(* PLC project CODEYS Common Library Template, TK TC6_v0200_Example1 v2.0, author 3S - Smart Software Solutions GmbH *)
(* stored: creationDateTime 2020-04-25T16:06:08.4861619, version 3.5.15.10, modificationDateTime 2020-04-25T16:01:39.8406952, organization 3S - Smart Software Solutions GmbH *)
(* Library project template with all possible element types, docu and a sample project structure *)

(* {attribute 'conditionalshow'} {attribute 'conditionalshow' := 'SomeText'} {attribute 'hide'} *)
{attribute 'qualified_only'}
TYPE ERROR : (NO_ERROR, TIME_OUT);
END_TYPE

{attribute 'qualified_only'}
VAR_GLOBAL CONSTANT  (* Constants - {attribute 'conditionalshow'} {attribute 'conditionalshow' := 'SomeText'} {attribute 'hide'} *)
  gc_iDummy : INT := 42;
END_VAR

{attribute 'qualified_only'}
VAR_GLOBAL  (* Variables - {attribute 'conditionalshow'} {attribute 'conditionalshow' := 'SomeText'} {attribute 'hide'} *)
  g_iDummy : INT;
END_VAR

(* {attribute 'hide_all_locals'} {attribute 'conditionalshow_all_locals' := 'SomeText'} {attribute 'conditionalshow_all_locals'} {attribute 'conditionalshow' := 'SomeText'} {attribute 'conditionalshow'} {attribute 'hide'} *)
FUNCTION_BLOCK ETrig_Temp EXTENDS CBML.ETrig
  VAR_OUTPUT
    eErrorID : ERROR;
  END_VAR

            SUPER^();
eErrorID := _Model.iErrorID;


          

METHOD CleanupAction
  VAR_INPUT
    xAbortProposed : BOOL;
    iErrorIDProposed : INT;
  END_VAR
  VAR_OUTPUT
    xComplete : BOOL := TRUE;
    xAbort : BOOL := xAbortProposed;
    iErrorID : INT := iErrorIDProposed;
  END_VAR
                  {analysis -2} 
/// ``CleanupAction`` is running until one of the following events occurs:
/// When ``xComplete`` is ``TRUE`` the state |STATE.DONE| is reached.
/// When ``xAbort`` is ``TRUE`` the state |STATE.ABORTED| is reached.
/// When ``iErrorID`` ≠ 0 (Zero) the state |STATE.ERROR| is reached.
///
/// | After a *Ready Condition* as input (``iErrorIDProposed`` = 0 and ``xAbortProposed`` = ``FALSE``), only the output states
/// | `DONE` (``xComplete`` is ``TRUE``) or `ERROR` (``iErrorID`` ≠ 0) are possible.
///
/// | After a *Error Condition* as input (``iErrorIDProposed`` ≠ 0), only the output state
/// | `ERROR` (``iErrorID`` ≠ 0) is possible.
///
/// | After a *Abort Condition* as Input (``xAbortProposed`` = ``TRUE``), only the output states
/// | `ABORTED` (``xAbort`` is ``TRUE``) or `ERROR` (``iErrorID`` ≠ 0) are possible.
///
/// .. admonition:: Example
///
///     .. code-block:: codesys
///     
///         (* common cleanup -- first steps *) 
///         
///         IF xComplete THEN
///             IF xAbortProposed THEN
///                 (* abort condition -- abort specific cleanup *)
///                 xAbort := TRUE;
///                 xComplete := FALSE;
///             ELSIF iErrorIDProposed <> 0 THEN
///                 (* error condition -- error specific cleanup *)
///                 iErrorID := SEL(xComplete, 0, iErrorIDProposed);
///                 xComplete := FALSE;
///             ELSE
///                 (* ready condition -- done specific cleanup*)
///             END_IF
///         END_IF
///
///         (* common cleanup -- last steps *) 
///
/// .. note::
///
///    If this method will not provide any implementation, please remove it!

                
END_METHOD

METHOD CyclicAction
  VAR_INPUT
    itfTimingController : CBML.ITimingController;
  END_VAR
  VAR_OUTPUT
    xComplete : BOOL := TRUE;
    iErrorID : INT := 0;
  END_VAR
                  {analysis -2} 
/// The CyclicAction is running until either ``xComplete`` is ``TRUE`` or ``iErrorID`` ≠  0 (Zero).
/// If ``xComplete`` is ``TRUE`` or ``iErrorID`` ≠  0 (Zero) the state |STATE.CLEANING| is reached.
/// With ``itfTimingController`` ≠  0 (Zero) it is possible to check the current invocation time (see: |ITimingController.ControllerCheckTiming|).
/// Function blocks with a ``udiTimeLimit`` input variable (see: |IETrigTl|, |IETrigATl|, |IETrigTlTo|, |IETrigATlTo|, |ILConTl|, |ILConTlTo|, |ILConTlC|)
/// should be implement in such a way that the current invocation is exited when the consumed time for this invocation has exceeded the settings from udiTimeLimit.
///
/// .. admonition:: Example
///
///     .. code-block:: codesys
///     
///         REPEAT
///             // working to reach the ready condition
///             // ⇒ xComplete := TRUE
///             // if the maximum invocation time is reached
///             // ⇒ xTimeLimit := TRUE
///             // if the maximum operating time is reached
///             // ⇒ xTimeOut := TRUE
///             // if an error condition is reached
///             // ⇒ set iErrorID to a value other than 0 (Zero)
///             itfTimingController.ControllerCheckTiming(
///                 xTimeOut=>xTimeOut,
///                 xTimeLimit=>xTimeLimit
///             );
///         
///             xComplete := TRUE;
///             iErrorID := ERROR.NO_ERROR;
///     
///         UNTIL xComplete OR
///               xTimeOut OR xTimeLimit OR
///               iErrorID <> ERROR.NO_ERROR
///         END_REPEAT
///
/// .. note::
///
///    If this method will not provide any implementation, please remove it!

                
END_METHOD

METHOD ExitAction
  VAR_INPUT
    xAfterCleanup : BOOL;
    xInCopyCode : BOOL;
  END_VAR
                  {analysis -2} 
/// This method is intended for releasing external resources (like RTS handles).
/// Do not call other internal function block instances in the context of this method.
/// Call only external functions defined inside the RTS.
/// For cleaning up other resources then external ones, please use the ``CleanupAction``.
/// This method should be callable in the context of ``FB_EXIT`` for example
/// before downloading a new application or before reseting an application.
///
/// .. note::
///
///    If this method will not provide any implementation, please remove it!

                
END_METHOD

METHOD ResetAction
  VAR_OUTPUT
    xComplete : BOOL := TRUE;
  END_VAR
                  {analysis -2} 
/// The ``ResetAction`` is running until the output ``xComplete`` is ``TRUE``.
/// If ``xComplete`` is ``TRUE`` the state |STATE.DORMANT| is reached.
///
/// .. note::
///
///    If this method will not provide any implementation, please remove it!

                
END_METHOD

METHOD SampleAction
  VAR_OUTPUT
    iErrorID : INT := 0;
  END_VAR
                  {analysis -2} 
/// After leaving the state |STATE.DORMANT| the ``SampleAction`` is running one time then the state |STATE.STARTING| is reached.
/// If there is a ``iErrorID`` ≠  0 (Zero) the state |STATE.CLEANING| is reached instead.
///
/// .. note::
///
///    If this method will not provide any implementation, please remove it!

                
END_METHOD

METHOD StartAction
  VAR_OUTPUT
    xComplete : BOOL := TRUE;
    iErrorID : INT := 0;
  END_VAR
                  {analysis -2} 
/// The ``StartAction`` is running until either the output ``xComplete`` is ``TRUE`` or ``iErrorID`` ≠ 0 (Zero).
/// If ``xComplete`` is ``TRUE`` the state |STATE.EXECUTING| is reached.
/// If there is a ``iErrorID`` ≠  0 (Zero) the state |STATE.CLEANING| is reached.
///
/// .. note::
///
///    To sample the inputs in the first invocation of a function block the method SampleAction is the solution of choice.
///    See: |ISampleActionProvider.SampleAction|
///
/// .. note::
///
///    If this method will not provide any implementation, please remove it!

                
END_METHOD
END_FUNCTION_BLOCK

(* {attribute 'hide_all_locals'} {attribute 'conditionalshow_all_locals' := 'SomeText'} {attribute 'conditionalshow_all_locals'} {attribute 'conditionalshow' := 'SomeText'} {attribute 'conditionalshow'} {attribute 'hide'} *)
FUNCTION_BLOCK ETrigA_Temp EXTENDS CBML.ETrigA
  VAR_OUTPUT
    eErrorID : ERROR;
  END_VAR

            SUPER^();
eErrorID := _Model.iErrorID;

          

METHOD CleanupAction
  VAR_INPUT
    xAbortProposed : BOOL;
    iErrorIDProposed : INT;
  END_VAR
  VAR_OUTPUT
    xComplete : BOOL := TRUE;
    xAbort : BOOL := xAbortProposed;
    iErrorID : INT := iErrorIDProposed;
  END_VAR
                  {analysis -2} 
/// ``CleanupAction`` is running until one of the following events occurs:
/// When ``xComplete`` is ``TRUE`` the state |STATE.DONE| is reached.
/// When ``xAbort`` is ``TRUE`` the state |STATE.ABORTED| is reached.
/// When ``iErrorID`` ≠ 0 (Zero) the state |STATE.ERROR| is reached.
///
/// | After a *Ready Condition* as input (``iErrorIDProposed`` = 0 and ``xAbortProposed`` = ``FALSE``), only the output states
/// | `DONE` (``xComplete`` is ``TRUE``) or `ERROR` (``iErrorID`` ≠ 0) are possible.
///
/// | After a *Error Condition* as input (``iErrorIDProposed`` ≠ 0), only the output state
/// | `ERROR` (``iErrorID`` ≠ 0) is possible.
///
/// | After a *Abort Condition* as Input (``xAbortProposed`` = ``TRUE``), only the output states
/// | `ABORTED` (``xAbort`` is ``TRUE``) or `ERROR` (``iErrorID`` ≠ 0) are possible.
///
/// .. admonition:: Example
///
///     .. code-block:: codesys
///     
///         (* common cleanup -- first steps *) 
///         
///         IF xComplete THEN
///             IF xAbortProposed THEN
///                 (* abort condition -- abort specific cleanup *)
///                 xAbort := TRUE;
///                 xComplete := FALSE;
///             ELSIF iErrorIDProposed <> 0 THEN
///                 (* error condition -- error specific cleanup *)
///                 iErrorID := SEL(xComplete, 0, iErrorIDProposed);
///                 xComplete := FALSE;
///             ELSE
///                 (* ready condition -- done specific cleanup*)
///             END_IF
///         END_IF
///
///         (* common cleanup -- last steps *) 
///
/// .. note::
///
///    If this method will not provide any implementation, please remove it!

                
END_METHOD

METHOD CyclicAction
  VAR_INPUT
    itfTimingController : CBML.ITimingController;
  END_VAR
  VAR_OUTPUT
    xComplete : BOOL := TRUE;
    iErrorID : INT := 0;
  END_VAR
                  {analysis -2} 
/// The CyclicAction is running until either ``xComplete`` is ``TRUE`` or ``iErrorID`` ≠  0 (Zero).
/// If ``xComplete`` is ``TRUE`` or ``iErrorID`` ≠  0 (Zero) the state |STATE.CLEANING| is reached.
/// With ``itfTimingController`` ≠  0 (Zero) it is possible to check the current invocation time (see: |ITimingController.ControllerCheckTiming|).
/// Function blocks with a ``udiTimeLimit`` input variable (see: |IETrigTl|, |IETrigATl|, |IETrigTlTo|, |IETrigATlTo|, |ILConTl|, |ILConTlTo|, |ILConTlC|)
/// should be implement in such a way that the current invocation is exited when the consumed time for this invocation has exceeded the settings from udiTimeLimit.
///
/// .. admonition:: Example
///
///     .. code-block:: codesys
///     
///         REPEAT
///             // working to reach the ready condition
///             // ⇒ xComplete := TRUE
///             // if the maximum invocation time is reached
///             // ⇒ xTimeLimit := TRUE
///             // if the maximum operating time is reached
///             // ⇒ xTimeOut := TRUE
///             // if an error condition is reached
///             // ⇒ set iErrorID to a value other than 0 (Zero)
///             itfTimingController.ControllerCheckTiming(
///                 xTimeOut=>xTimeOut,
///                 xTimeLimit=>xTimeLimit
///             );
///         
///             xComplete := TRUE;
///             iErrorID := ERROR.NO_ERROR;
///     
///         UNTIL xComplete OR
///               xTimeOut OR xTimeLimit OR
///               iErrorID <> ERROR.NO_ERROR
///         END_REPEAT
///
/// .. note::
///
///    If this method will not provide any implementation, please remove it!

                
END_METHOD

METHOD ExitAction
  VAR_INPUT
    xAfterCleanup : BOOL;
    xInCopyCode : BOOL;
  END_VAR
                  {analysis -2} 
/// This method is intended for releasing external resources (like RTS handles).
/// Do not call other internal function block instances in the context of this method.
/// Call only external functions defined inside the RTS.
/// For cleaning up other resources then external ones, please use the ``CleanupAction``.
/// This method should be callable in the context of ``FB_EXIT`` for example
/// before downloading a new application or before reseting an application.
///
/// .. note::
///
///    If this method will not provide any implementation, please remove it!

                
END_METHOD

METHOD ResetAction
  VAR_OUTPUT
    xComplete : BOOL := TRUE;
  END_VAR
                  {analysis -2} 
/// The ``ResetAction`` is running until the output ``xComplete`` is ``TRUE``.
/// If ``xComplete`` is ``TRUE`` the state |STATE.DORMANT| is reached.
///
/// .. note::
///
///    If this method will not provide any implementation, please remove it!

                
END_METHOD

METHOD SampleAction
  VAR_OUTPUT
    iErrorID : INT := 0;
  END_VAR
                  {analysis -2} 
/// After leaving the state |STATE.DORMANT| the ``SampleAction`` is running one time then the state |STATE.STARTING| is reached.
/// If there is a ``iErrorID`` ≠  0 (Zero) the state |STATE.CLEANING| is reached instead.
///
/// .. note::
///
///    If this method will not provide any implementation, please remove it!

                
END_METHOD

METHOD StartAction
  VAR_OUTPUT
    xComplete : BOOL := TRUE;
    iErrorID : INT := 0;
  END_VAR
                  {analysis -2} 
/// The ``StartAction`` is running until either the output ``xComplete`` is ``TRUE`` or ``iErrorID`` ≠ 0 (Zero).
/// If ``xComplete`` is ``TRUE`` the state |STATE.EXECUTING| is reached.
/// If there is a ``iErrorID`` ≠  0 (Zero) the state |STATE.CLEANING| is reached.
///
/// .. note::
///
///    To sample the inputs in the first invocation of a function block the method SampleAction is the solution of choice.
///    See: |ISampleActionProvider.SampleAction|
///
/// .. note::
///
///    If this method will not provide any implementation, please remove it!

                
END_METHOD
END_FUNCTION_BLOCK

(* {attribute 'hide_all_locals'} {attribute 'conditionalshow_all_locals' := 'SomeText'} {attribute 'conditionalshow_all_locals'} {attribute 'conditionalshow' := 'SomeText'} {attribute 'conditionalshow'} {attribute 'hide'} *)
FUNCTION_BLOCK ETrigATl_Temp EXTENDS CBML.ETrigATl
  VAR_OUTPUT
    eErrorID : ERROR;
  END_VAR

            SUPER^();
eErrorID := _Model.iErrorID;

          

METHOD CleanupAction
  VAR_INPUT
    xAbortProposed : BOOL;
    iErrorIDProposed : INT;
  END_VAR
  VAR_OUTPUT
    xComplete : BOOL := TRUE;
    xAbort : BOOL := xAbortProposed;
    iErrorID : INT := iErrorIDProposed;
  END_VAR
                  {analysis -2} 
/// ``CleanupAction`` is running until one of the following events occurs:
/// When ``xComplete`` is ``TRUE`` the state |STATE.DONE| is reached.
/// When ``xAbort`` is ``TRUE`` the state |STATE.ABORTED| is reached.
/// When ``iErrorID`` ≠ 0 (Zero) the state |STATE.ERROR| is reached.
///
/// | After a *Ready Condition* as input (``iErrorIDProposed`` = 0 and ``xAbortProposed`` = ``FALSE``), only the output states
/// | `DONE` (``xComplete`` is ``TRUE``) or `ERROR` (``iErrorID`` ≠ 0) are possible.
///
/// | After a *Error Condition* as input (``iErrorIDProposed`` ≠ 0), only the output state
/// | `ERROR` (``iErrorID`` ≠ 0) is possible.
///
/// | After a *Abort Condition* as Input (``xAbortProposed`` = ``TRUE``), only the output states
/// | `ABORTED` (``xAbort`` is ``TRUE``) or `ERROR` (``iErrorID`` ≠ 0) are possible.
///
/// .. admonition:: Example
///
///     .. code-block:: codesys
///     
///         (* common cleanup -- first steps *) 
///         
///         IF xComplete THEN
///             IF xAbortProposed THEN
///                 (* abort condition -- abort specific cleanup *)
///                 xAbort := TRUE;
///                 xComplete := FALSE;
///             ELSIF iErrorIDProposed <> 0 THEN
///                 (* error condition -- error specific cleanup *)
///                 iErrorID := SEL(xComplete, 0, iErrorIDProposed);
///                 xComplete := FALSE;
///             ELSE
///                 (* ready condition -- done specific cleanup*)
///             END_IF
///         END_IF
///
///         (* common cleanup -- last steps *) 
///
/// .. note::
///
///    If this method will not provide any implementation, please remove it!

                
END_METHOD

METHOD CyclicAction
  VAR_INPUT
    itfTimingController : CBML.ITimingController;
  END_VAR
  VAR_OUTPUT
    xComplete : BOOL := TRUE;
    iErrorID : INT := 0;
  END_VAR
                  {analysis -2} 
/// The CyclicAction is running until either ``xComplete`` is ``TRUE`` or ``iErrorID`` ≠  0 (Zero).
/// If ``xComplete`` is ``TRUE`` or ``iErrorID`` ≠  0 (Zero) the state |STATE.CLEANING| is reached.
/// With ``itfTimingController`` ≠  0 (Zero) it is possible to check the current invocation time (see: |ITimingController.ControllerCheckTiming|).
/// Function blocks with a ``udiTimeLimit`` input variable (see: |IETrigTl|, |IETrigATl|, |IETrigTlTo|, |IETrigATlTo|, |ILConTl|, |ILConTlTo|, |ILConTlC|)
/// should be implement in such a way that the current invocation is exited when the consumed time for this invocation has exceeded the settings from udiTimeLimit.
///
/// .. admonition:: Example
///
///     .. code-block:: codesys
///     
///         REPEAT
///             // working to reach the ready condition
///             // ⇒ xComplete := TRUE
///             // if the maximum invocation time is reached
///             // ⇒ xTimeLimit := TRUE
///             // if the maximum operating time is reached
///             // ⇒ xTimeOut := TRUE
///             // if an error condition is reached
///             // ⇒ set iErrorID to a value other than 0 (Zero)
///             itfTimingController.ControllerCheckTiming(
///                 xTimeOut=>xTimeOut,
///                 xTimeLimit=>xTimeLimit
///             );
///         
///             xComplete := TRUE;
///             iErrorID := ERROR.NO_ERROR;
///     
///         UNTIL xComplete OR
///               xTimeOut OR xTimeLimit OR
///               iErrorID <> ERROR.NO_ERROR
///         END_REPEAT
///
/// .. note::
///
///    If this method will not provide any implementation, please remove it!

                
END_METHOD

METHOD ExitAction
  VAR_INPUT
    xAfterCleanup : BOOL;
    xInCopyCode : BOOL;
  END_VAR
                  {analysis -2} 
/// This method is intended for releasing external resources (like RTS handles).
/// Do not call other internal function block instances in the context of this method.
/// Call only external functions defined inside the RTS.
/// For cleaning up other resources then external ones, please use the ``CleanupAction``.
/// This method should be callable in the context of ``FB_EXIT`` for example
/// before downloading a new application or before reseting an application.
///
/// .. note::
///
///    If this method will not provide any implementation, please remove it!

                
END_METHOD

METHOD ResetAction
  VAR_OUTPUT
    xComplete : BOOL := TRUE;
  END_VAR
                  {analysis -2} 
/// The ``ResetAction`` is running until the output ``xComplete`` is ``TRUE``.
/// If ``xComplete`` is ``TRUE`` the state |STATE.DORMANT| is reached.
///
/// .. note::
///
///    If this method will not provide any implementation, please remove it!

                
END_METHOD

METHOD SampleAction
  VAR_OUTPUT
    iErrorID : INT := 0;
  END_VAR
                  {analysis -2} 
/// After leaving the state |STATE.DORMANT| the ``SampleAction`` is running one time then the state |STATE.STARTING| is reached.
/// If there is a ``iErrorID`` ≠  0 (Zero) the state |STATE.CLEANING| is reached instead.
///
/// .. note::
///
///    If this method will not provide any implementation, please remove it!

                
END_METHOD

METHOD StartAction
  VAR_OUTPUT
    xComplete : BOOL := TRUE;
    iErrorID : INT := 0;
  END_VAR
                  {analysis -2} 
/// The ``StartAction`` is running until either the output ``xComplete`` is ``TRUE`` or ``iErrorID`` ≠ 0 (Zero).
/// If ``xComplete`` is ``TRUE`` the state |STATE.EXECUTING| is reached.
/// If there is a ``iErrorID`` ≠  0 (Zero) the state |STATE.CLEANING| is reached.
///
/// .. note::
///
///    To sample the inputs in the first invocation of a function block the method SampleAction is the solution of choice.
///    See: |ISampleActionProvider.SampleAction|
///
/// .. note::
///
///    If this method will not provide any implementation, please remove it!

                
END_METHOD
END_FUNCTION_BLOCK

(* {attribute 'hide_all_locals'} {attribute 'conditionalshow_all_locals' := 'SomeText'} {attribute 'conditionalshow_all_locals'} {attribute 'conditionalshow' := 'SomeText'} {attribute 'conditionalshow'} {attribute 'hide'} *)
FUNCTION_BLOCK ETrigATlTo_Temp EXTENDS CBML.ETrigATlTo
  VAR_OUTPUT
    eErrorID : ERROR;  (* specific Outputs *)
  END_VAR

            SUPER^();
IF _Model.iErrorID = CBML.ERROR.TIME_OUT THEN
	eErrorID := ERROR.TIME_OUT;
ELSE
	eErrorID := _Model.iErrorID;
END_IF

          

METHOD CleanupAction
  VAR_INPUT
    xAbortProposed : BOOL;
    iErrorIDProposed : INT;
  END_VAR
  VAR_OUTPUT
    xComplete : BOOL := TRUE;
    xAbort : BOOL := xAbortProposed;
    iErrorID : INT := iErrorIDProposed;
  END_VAR
                  {analysis -2} 
/// ``CleanupAction`` is running until one of the following events occurs:
/// When ``xComplete`` is ``TRUE`` the state |STATE.DONE| is reached.
/// When ``xAbort`` is ``TRUE`` the state |STATE.ABORTED| is reached.
/// When ``iErrorID`` ≠ 0 (Zero) the state |STATE.ERROR| is reached.
///
/// | After a *Ready Condition* as input (``iErrorIDProposed`` = 0 and ``xAbortProposed`` = ``FALSE``), only the output states
/// | `DONE` (``xComplete`` is ``TRUE``) or `ERROR` (``iErrorID`` ≠ 0) are possible.
///
/// | After a *Error Condition* as input (``iErrorIDProposed`` ≠ 0), only the output state
/// | `ERROR` (``iErrorID`` ≠ 0) is possible.
///
/// | After a *Abort Condition* as Input (``xAbortProposed`` = ``TRUE``), only the output states
/// | `ABORTED` (``xAbort`` is ``TRUE``) or `ERROR` (``iErrorID`` ≠ 0) are possible.
///
/// .. admonition:: Example
///
///     .. code-block:: codesys
///     
///         (* common cleanup -- first steps *) 
///         
///         IF xComplete THEN
///             IF xAbortProposed THEN
///                 (* abort condition -- abort specific cleanup *)
///                 xAbort := TRUE;
///                 xComplete := FALSE;
///             ELSIF iErrorIDProposed <> 0 THEN
///                 (* error condition -- error specific cleanup *)
///                 iErrorID := SEL(xComplete, 0, iErrorIDProposed);
///                 xComplete := FALSE;
///             ELSE
///                 (* ready condition -- done specific cleanup*)
///             END_IF
///         END_IF
///
///         (* common cleanup -- last steps *) 
///
/// .. note::
///
///    If this method will not provide any implementation, please remove it!

                
END_METHOD

METHOD CyclicAction
  VAR_INPUT
    itfTimingController : CBML.ITimingController;
  END_VAR
  VAR_OUTPUT
    xComplete : BOOL := TRUE;
    iErrorID : INT := 0;
  END_VAR
                  {analysis -2} 
/// The CyclicAction is running until either ``xComplete`` is ``TRUE`` or ``iErrorID`` ≠  0 (Zero).
/// If ``xComplete`` is ``TRUE`` or ``iErrorID`` ≠  0 (Zero) the state |STATE.CLEANING| is reached.
/// With ``itfTimingController`` ≠  0 (Zero) it is possible to check the current invocation time (see: |ITimingController.ControllerCheckTiming|).
/// Function blocks with a ``udiTimeLimit`` input variable (see: |IETrigTl|, |IETrigATl|, |IETrigTlTo|, |IETrigATlTo|, |ILConTl|, |ILConTlTo|, |ILConTlC|)
/// should be implement in such a way that the current invocation is exited when the consumed time for this invocation has exceeded the settings from udiTimeLimit.
///
/// .. admonition:: Example
///
///     .. code-block:: codesys
///     
///         REPEAT
///             // working to reach the ready condition
///             // ⇒ xComplete := TRUE
///             // if the maximum invocation time is reached
///             // ⇒ xTimeLimit := TRUE
///             // if the maximum operating time is reached
///             // ⇒ xTimeOut := TRUE
///             // if an error condition is reached
///             // ⇒ set iErrorID to a value other than 0 (Zero)
///             itfTimingController.ControllerCheckTiming(
///                 xTimeOut=>xTimeOut,
///                 xTimeLimit=>xTimeLimit
///             );
///         
///             xComplete := TRUE;
///             iErrorID := ERROR.NO_ERROR;
///     
///         UNTIL xComplete OR
///               xTimeOut OR xTimeLimit OR
///               iErrorID <> ERROR.NO_ERROR
///         END_REPEAT
///
/// .. note::
///
///    If this method will not provide any implementation, please remove it!

                
END_METHOD

METHOD ExitAction
  VAR_INPUT
    xAfterCleanup : BOOL;
    xInCopyCode : BOOL;
  END_VAR
                  {analysis -2} 
/// This method is intended for releasing external resources (like RTS handles).
/// Do not call other internal function block instances in the context of this method.
/// Call only external functions defined inside the RTS.
/// For cleaning up other resources then external ones, please use the ``CleanupAction``.
/// This method should be callable in the context of ``FB_EXIT`` for example
/// before downloading a new application or before reseting an application.
///
/// .. note::
///
///    If this method will not provide any implementation, please remove it!

                
END_METHOD

METHOD ResetAction
  VAR_OUTPUT
    xComplete : BOOL := TRUE;
  END_VAR
                  {analysis -2} 
/// The ``ResetAction`` is running until the output ``xComplete`` is ``TRUE``.
/// If ``xComplete`` is ``TRUE`` the state |STATE.DORMANT| is reached.
///
/// .. note::
///
///    If this method will not provide any implementation, please remove it!

                
END_METHOD

METHOD SampleAction
  VAR_OUTPUT
    iErrorID : INT := 0;
  END_VAR
                  {analysis -2} 
/// After leaving the state |STATE.DORMANT| the ``SampleAction`` is running one time then the state |STATE.STARTING| is reached.
/// If there is a ``iErrorID`` ≠  0 (Zero) the state |STATE.CLEANING| is reached instead.
///
/// .. note::
///
///    If this method will not provide any implementation, please remove it!

                
END_METHOD

METHOD StartAction
  VAR_OUTPUT
    xComplete : BOOL := TRUE;
    iErrorID : INT := 0;
  END_VAR
                  {analysis -2} 
/// The ``StartAction`` is running until either the output ``xComplete`` is ``TRUE`` or ``iErrorID`` ≠ 0 (Zero).
/// If ``xComplete`` is ``TRUE`` the state |STATE.EXECUTING| is reached.
/// If there is a ``iErrorID`` ≠  0 (Zero) the state |STATE.CLEANING| is reached.
///
/// .. note::
///
///    To sample the inputs in the first invocation of a function block the method SampleAction is the solution of choice.
///    See: |ISampleActionProvider.SampleAction|
///
/// .. note::
///
///    If this method will not provide any implementation, please remove it!

                
END_METHOD
END_FUNCTION_BLOCK

(* {attribute 'hide_all_locals'} {attribute 'conditionalshow_all_locals' := 'SomeText'} {attribute 'conditionalshow_all_locals'} {attribute 'conditionalshow' := 'SomeText'} {attribute 'conditionalshow'} {attribute 'hide'} *)
FUNCTION_BLOCK ETrigATo_Temp EXTENDS CBML.ETrigATo
  VAR_OUTPUT
    eErrorID : ERROR;
  END_VAR

            SUPER^();
IF _Model.iErrorID = CBML.ERROR.TIME_OUT THEN
	eErrorID := ERROR.TIME_OUT;
ELSE
	eErrorID := _Model.iErrorID;
END_IF

          

METHOD CleanupAction
  VAR_INPUT
    xAbortProposed : BOOL;
    iErrorIDProposed : INT;
  END_VAR
  VAR_OUTPUT
    xComplete : BOOL := TRUE;
    xAbort : BOOL := xAbortProposed;
    iErrorID : INT := iErrorIDProposed;
  END_VAR
                  {analysis -2} 
/// ``CleanupAction`` is running until one of the following events occurs:
/// When ``xComplete`` is ``TRUE`` the state |STATE.DONE| is reached.
/// When ``xAbort`` is ``TRUE`` the state |STATE.ABORTED| is reached.
/// When ``iErrorID`` ≠ 0 (Zero) the state |STATE.ERROR| is reached.
///
/// | After a *Ready Condition* as input (``iErrorIDProposed`` = 0 and ``xAbortProposed`` = ``FALSE``), only the output states
/// | `DONE` (``xComplete`` is ``TRUE``) or `ERROR` (``iErrorID`` ≠ 0) are possible.
///
/// | After a *Error Condition* as input (``iErrorIDProposed`` ≠ 0), only the output state
/// | `ERROR` (``iErrorID`` ≠ 0) is possible.
///
/// | After a *Abort Condition* as Input (``xAbortProposed`` = ``TRUE``), only the output states
/// | `ABORTED` (``xAbort`` is ``TRUE``) or `ERROR` (``iErrorID`` ≠ 0) are possible.
///
/// .. admonition:: Example
///
///     .. code-block:: codesys
///     
///         (* common cleanup -- first steps *) 
///         
///         IF xComplete THEN
///             IF xAbortProposed THEN
///                 (* abort condition -- abort specific cleanup *)
///                 xAbort := TRUE;
///                 xComplete := FALSE;
///             ELSIF iErrorIDProposed <> 0 THEN
///                 (* error condition -- error specific cleanup *)
///                 iErrorID := SEL(xComplete, 0, iErrorIDProposed);
///                 xComplete := FALSE;
///             ELSE
///                 (* ready condition -- done specific cleanup*)
///             END_IF
///         END_IF
///
///         (* common cleanup -- last steps *) 
///
/// .. note::
///
///    If this method will not provide any implementation, please remove it!

                
END_METHOD

METHOD CyclicAction
  VAR_INPUT
    itfTimingController : CBML.ITimingController;
  END_VAR
  VAR_OUTPUT
    xComplete : BOOL := TRUE;
    iErrorID : INT := 0;
  END_VAR
                  {analysis -2} 
/// The CyclicAction is running until either ``xComplete`` is ``TRUE`` or ``iErrorID`` ≠  0 (Zero).
/// If ``xComplete`` is ``TRUE`` or ``iErrorID`` ≠  0 (Zero) the state |STATE.CLEANING| is reached.
/// With ``itfTimingController`` ≠  0 (Zero) it is possible to check the current invocation time (see: |ITimingController.ControllerCheckTiming|).
/// Function blocks with a ``udiTimeLimit`` input variable (see: |IETrigTl|, |IETrigATl|, |IETrigTlTo|, |IETrigATlTo|, |ILConTl|, |ILConTlTo|, |ILConTlC|)
/// should be implement in such a way that the current invocation is exited when the consumed time for this invocation has exceeded the settings from udiTimeLimit.
///
/// .. admonition:: Example
///
///     .. code-block:: codesys
///     
///         REPEAT
///             // working to reach the ready condition
///             // ⇒ xComplete := TRUE
///             // if the maximum invocation time is reached
///             // ⇒ xTimeLimit := TRUE
///             // if the maximum operating time is reached
///             // ⇒ xTimeOut := TRUE
///             // if an error condition is reached
///             // ⇒ set iErrorID to a value other than 0 (Zero)
///             itfTimingController.ControllerCheckTiming(
///                 xTimeOut=>xTimeOut,
///                 xTimeLimit=>xTimeLimit
///             );
///         
///             xComplete := TRUE;
///             iErrorID := ERROR.NO_ERROR;
///     
///         UNTIL xComplete OR
///               xTimeOut OR xTimeLimit OR
///               iErrorID <> ERROR.NO_ERROR
///         END_REPEAT
///
/// .. note::
///
///    If this method will not provide any implementation, please remove it!

                
END_METHOD

METHOD ExitAction
  VAR_INPUT
    xAfterCleanup : BOOL;
    xInCopyCode : BOOL;
  END_VAR
                  {analysis -2} 
/// This method is intended for releasing external resources (like RTS handles).
/// Do not call other internal function block instances in the context of this method.
/// Call only external functions defined inside the RTS.
/// For cleaning up other resources then external ones, please use the ``CleanupAction``.
/// This method should be callable in the context of ``FB_EXIT`` for example
/// before downloading a new application or before reseting an application.
///
/// .. note::
///
///    If this method will not provide any implementation, please remove it!

                
END_METHOD

METHOD ResetAction
  VAR_OUTPUT
    xComplete : BOOL := TRUE;
  END_VAR
                  {analysis -2} 
/// The ``ResetAction`` is running until the output ``xComplete`` is ``TRUE``.
/// If ``xComplete`` is ``TRUE`` the state |STATE.DORMANT| is reached.
///
/// .. note::
///
///    If this method will not provide any implementation, please remove it!

                
END_METHOD

METHOD SampleAction
  VAR_OUTPUT
    iErrorID : INT := 0;
  END_VAR
                  {analysis -2} 
/// After leaving the state |STATE.DORMANT| the ``SampleAction`` is running one time then the state |STATE.STARTING| is reached.
/// If there is a ``iErrorID`` ≠  0 (Zero) the state |STATE.CLEANING| is reached instead.
///
/// .. note::
///
///    If this method will not provide any implementation, please remove it!

                
END_METHOD

METHOD StartAction
  VAR_OUTPUT
    xComplete : BOOL := TRUE;
    iErrorID : INT := 0;
  END_VAR
                  {analysis -2} 
/// The ``StartAction`` is running until either the output ``xComplete`` is ``TRUE`` or ``iErrorID`` ≠ 0 (Zero).
/// If ``xComplete`` is ``TRUE`` the state |STATE.EXECUTING| is reached.
/// If there is a ``iErrorID`` ≠  0 (Zero) the state |STATE.CLEANING| is reached.
///
/// .. note::
///
///    To sample the inputs in the first invocation of a function block the method SampleAction is the solution of choice.
///    See: |ISampleActionProvider.SampleAction|
///
/// .. note::
///
///    If this method will not provide any implementation, please remove it!

                
END_METHOD
END_FUNCTION_BLOCK

(* {attribute 'hide_all_locals'} {attribute 'conditionalshow_all_locals' := 'SomeText'} {attribute 'conditionalshow_all_locals'} {attribute 'conditionalshow' := 'SomeText'} {attribute 'conditionalshow'} {attribute 'hide'} *)
FUNCTION_BLOCK ETrigTl_Temp EXTENDS CBML.ETrigTl
  VAR_OUTPUT
    eErrorID : ERROR;
  END_VAR

            SUPER^();
eErrorID := _Model.iErrorID;

          

METHOD CleanupAction
  VAR_INPUT
    xAbortProposed : BOOL;
    iErrorIDProposed : INT;
  END_VAR
  VAR_OUTPUT
    xComplete : BOOL := TRUE;
    xAbort : BOOL := xAbortProposed;
    iErrorID : INT := iErrorIDProposed;
  END_VAR
                  {analysis -2} 
/// ``CleanupAction`` is running until one of the following events occurs:
/// When ``xComplete`` is ``TRUE`` the state |STATE.DONE| is reached.
/// When ``xAbort`` is ``TRUE`` the state |STATE.ABORTED| is reached.
/// When ``iErrorID`` ≠ 0 (Zero) the state |STATE.ERROR| is reached.
///
/// | After a *Ready Condition* as input (``iErrorIDProposed`` = 0 and ``xAbortProposed`` = ``FALSE``), only the output states
/// | `DONE` (``xComplete`` is ``TRUE``) or `ERROR` (``iErrorID`` ≠ 0) are possible.
///
/// | After a *Error Condition* as input (``iErrorIDProposed`` ≠ 0), only the output state
/// | `ERROR` (``iErrorID`` ≠ 0) is possible.
///
/// | After a *Abort Condition* as Input (``xAbortProposed`` = ``TRUE``), only the output states
/// | `ABORTED` (``xAbort`` is ``TRUE``) or `ERROR` (``iErrorID`` ≠ 0) are possible.
///
/// .. admonition:: Example
///
///     .. code-block:: codesys
///     
///         (* common cleanup -- first steps *) 
///         
///         IF xComplete THEN
///             IF xAbortProposed THEN
///                 (* abort condition -- abort specific cleanup *)
///                 xAbort := TRUE;
///                 xComplete := FALSE;
///             ELSIF iErrorIDProposed <> 0 THEN
///                 (* error condition -- error specific cleanup *)
///                 iErrorID := SEL(xComplete, 0, iErrorIDProposed);
///                 xComplete := FALSE;
///             ELSE
///                 (* ready condition -- done specific cleanup*)
///             END_IF
///         END_IF
///
///         (* common cleanup -- last steps *) 
///
/// .. note::
///
///    If this method will not provide any implementation, please remove it!

                
END_METHOD

METHOD CyclicAction
  VAR_INPUT
    itfTimingController : CBML.ITimingController;
  END_VAR
  VAR_OUTPUT
    xComplete : BOOL := TRUE;
    iErrorID : INT := 0;
  END_VAR
                  {analysis -2} 
/// The CyclicAction is running until either ``xComplete`` is ``TRUE`` or ``iErrorID`` ≠  0 (Zero).
/// If ``xComplete`` is ``TRUE`` or ``iErrorID`` ≠  0 (Zero) the state |STATE.CLEANING| is reached.
/// With ``itfTimingController`` ≠  0 (Zero) it is possible to check the current invocation time (see: |ITimingController.ControllerCheckTiming|).
/// Function blocks with a ``udiTimeLimit`` input variable (see: |IETrigTl|, |IETrigATl|, |IETrigTlTo|, |IETrigATlTo|, |ILConTl|, |ILConTlTo|, |ILConTlC|)
/// should be implement in such a way that the current invocation is exited when the consumed time for this invocation has exceeded the settings from udiTimeLimit.
///
/// .. admonition:: Example
///
///     .. code-block:: codesys
///     
///         REPEAT
///             // working to reach the ready condition
///             // ⇒ xComplete := TRUE
///             // if the maximum invocation time is reached
///             // ⇒ xTimeLimit := TRUE
///             // if the maximum operating time is reached
///             // ⇒ xTimeOut := TRUE
///             // if an error condition is reached
///             // ⇒ set iErrorID to a value other than 0 (Zero)
///             itfTimingController.ControllerCheckTiming(
///                 xTimeOut=>xTimeOut,
///                 xTimeLimit=>xTimeLimit
///             );
///         
///             xComplete := TRUE;
///             iErrorID := ERROR.NO_ERROR;
///     
///         UNTIL xComplete OR
///               xTimeOut OR xTimeLimit OR
///               iErrorID <> ERROR.NO_ERROR
///         END_REPEAT
///
/// .. note::
///
///    If this method will not provide any implementation, please remove it!

                
END_METHOD

METHOD ExitAction
  VAR_INPUT
    xAfterCleanup : BOOL;
    xInCopyCode : BOOL;
  END_VAR
                  {analysis -2} 
/// This method is intended for releasing external resources (like RTS handles).
/// Do not call other internal function block instances in the context of this method.
/// Call only external functions defined inside the RTS.
/// For cleaning up other resources then external ones, please use the ``CleanupAction``.
/// This method should be callable in the context of ``FB_EXIT`` for example
/// before downloading a new application or before reseting an application.
///
/// .. note::
///
///    If this method will not provide any implementation, please remove it!

                
END_METHOD

METHOD ResetAction
  VAR_OUTPUT
    xComplete : BOOL := TRUE;
  END_VAR
                  {analysis -2} 
/// The ``ResetAction`` is running until the output ``xComplete`` is ``TRUE``.
/// If ``xComplete`` is ``TRUE`` the state |STATE.DORMANT| is reached.
///
/// .. note::
///
///    If this method will not provide any implementation, please remove it!

                
END_METHOD

METHOD SampleAction
  VAR_OUTPUT
    iErrorID : INT := 0;
  END_VAR
                  {analysis -2} 
/// After leaving the state |STATE.DORMANT| the ``SampleAction`` is running one time then the state |STATE.STARTING| is reached.
/// If there is a ``iErrorID`` ≠  0 (Zero) the state |STATE.CLEANING| is reached instead.
///
/// .. note::
///
///    If this method will not provide any implementation, please remove it!

                
END_METHOD

METHOD StartAction
  VAR_OUTPUT
    xComplete : BOOL := TRUE;
    iErrorID : INT := 0;
  END_VAR
                  {analysis -2} 
/// The ``StartAction`` is running until either the output ``xComplete`` is ``TRUE`` or ``iErrorID`` ≠ 0 (Zero).
/// If ``xComplete`` is ``TRUE`` the state |STATE.EXECUTING| is reached.
/// If there is a ``iErrorID`` ≠  0 (Zero) the state |STATE.CLEANING| is reached.
///
/// .. note::
///
///    To sample the inputs in the first invocation of a function block the method SampleAction is the solution of choice.
///    See: |ISampleActionProvider.SampleAction|
///
/// .. note::
///
///    If this method will not provide any implementation, please remove it!

                
END_METHOD
END_FUNCTION_BLOCK

(* {attribute 'hide_all_locals'} {attribute 'conditionalshow_all_locals' := 'SomeText'} {attribute 'conditionalshow_all_locals'} {attribute 'conditionalshow' := 'SomeText'} {attribute 'conditionalshow'} {attribute 'hide'} *)
FUNCTION_BLOCK ETrigTlTo_Temp EXTENDS CBML.ETrigTlTo
  VAR_OUTPUT
    eErrorID : ERROR;
  END_VAR

            SUPER^();
IF _Model.iErrorID = CBML.ERROR.TIME_OUT THEN
	eErrorID := ERROR.TIME_OUT;
ELSE
	eErrorID := _Model.iErrorID;
END_IF

          

METHOD CleanupAction
  VAR_INPUT
    xAbortProposed : BOOL;
    iErrorIDProposed : INT;
  END_VAR
  VAR_OUTPUT
    xComplete : BOOL := TRUE;
    xAbort : BOOL := xAbortProposed;
    iErrorID : INT := iErrorIDProposed;
  END_VAR
                  {analysis -2} 
/// ``CleanupAction`` is running until one of the following events occurs:
/// When ``xComplete`` is ``TRUE`` the state |STATE.DONE| is reached.
/// When ``xAbort`` is ``TRUE`` the state |STATE.ABORTED| is reached.
/// When ``iErrorID`` ≠ 0 (Zero) the state |STATE.ERROR| is reached.
///
/// | After a *Ready Condition* as input (``iErrorIDProposed`` = 0 and ``xAbortProposed`` = ``FALSE``), only the output states
/// | `DONE` (``xComplete`` is ``TRUE``) or `ERROR` (``iErrorID`` ≠ 0) are possible.
///
/// | After a *Error Condition* as input (``iErrorIDProposed`` ≠ 0), only the output state
/// | `ERROR` (``iErrorID`` ≠ 0) is possible.
///
/// | After a *Abort Condition* as Input (``xAbortProposed`` = ``TRUE``), only the output states
/// | `ABORTED` (``xAbort`` is ``TRUE``) or `ERROR` (``iErrorID`` ≠ 0) are possible.
///
/// .. admonition:: Example
///
///     .. code-block:: codesys
///     
///         (* common cleanup -- first steps *) 
///         
///         IF xComplete THEN
///             IF xAbortProposed THEN
///                 (* abort condition -- abort specific cleanup *)
///                 xAbort := TRUE;
///                 xComplete := FALSE;
///             ELSIF iErrorIDProposed <> 0 THEN
///                 (* error condition -- error specific cleanup *)
///                 iErrorID := SEL(xComplete, 0, iErrorIDProposed);
///                 xComplete := FALSE;
///             ELSE
///                 (* ready condition -- done specific cleanup*)
///             END_IF
///         END_IF
///
///         (* common cleanup -- last steps *) 
///
/// .. note::
///
///    If this method will not provide any implementation, please remove it!

                
END_METHOD

METHOD CyclicAction
  VAR_INPUT
    itfTimingController : CBML.ITimingController;
  END_VAR
  VAR_OUTPUT
    xComplete : BOOL := TRUE;
    iErrorID : INT := 0;
  END_VAR
                  {analysis -2} 
/// The CyclicAction is running until either ``xComplete`` is ``TRUE`` or ``iErrorID`` ≠  0 (Zero).
/// If ``xComplete`` is ``TRUE`` or ``iErrorID`` ≠  0 (Zero) the state |STATE.CLEANING| is reached.
/// With ``itfTimingController`` ≠  0 (Zero) it is possible to check the current invocation time (see: |ITimingController.ControllerCheckTiming|).
/// Function blocks with a ``udiTimeLimit`` input variable (see: |IETrigTl|, |IETrigATl|, |IETrigTlTo|, |IETrigATlTo|, |ILConTl|, |ILConTlTo|, |ILConTlC|)
/// should be implement in such a way that the current invocation is exited when the consumed time for this invocation has exceeded the settings from udiTimeLimit.
///
/// .. admonition:: Example
///
///     .. code-block:: codesys
///     
///         REPEAT
///             // working to reach the ready condition
///             // ⇒ xComplete := TRUE
///             // if the maximum invocation time is reached
///             // ⇒ xTimeLimit := TRUE
///             // if the maximum operating time is reached
///             // ⇒ xTimeOut := TRUE
///             // if an error condition is reached
///             // ⇒ set iErrorID to a value other than 0 (Zero)
///             itfTimingController.ControllerCheckTiming(
///                 xTimeOut=>xTimeOut,
///                 xTimeLimit=>xTimeLimit
///             );
///         
///             xComplete := TRUE;
///             iErrorID := ERROR.NO_ERROR;
///     
///         UNTIL xComplete OR
///               xTimeOut OR xTimeLimit OR
///               iErrorID <> ERROR.NO_ERROR
///         END_REPEAT
///
/// .. note::
///
///    If this method will not provide any implementation, please remove it!

                
END_METHOD

METHOD ExitAction
  VAR_INPUT
    xAfterCleanup : BOOL;
    xInCopyCode : BOOL;
  END_VAR
                  {analysis -2} 
/// This method is intended for releasing external resources (like RTS handles).
/// Do not call other internal function block instances in the context of this method.
/// Call only external functions defined inside the RTS.
/// For cleaning up other resources then external ones, please use the ``CleanupAction``.
/// This method should be callable in the context of ``FB_EXIT`` for example
/// before downloading a new application or before reseting an application.
///
/// .. note::
///
///    If this method will not provide any implementation, please remove it!

                
END_METHOD

METHOD ResetAction
  VAR_OUTPUT
    xComplete : BOOL := TRUE;
  END_VAR
                  {analysis -2} 
/// The ``ResetAction`` is running until the output ``xComplete`` is ``TRUE``.
/// If ``xComplete`` is ``TRUE`` the state |STATE.DORMANT| is reached.
///
/// .. note::
///
///    If this method will not provide any implementation, please remove it!

                
END_METHOD

METHOD SampleAction
  VAR_OUTPUT
    iErrorID : INT := 0;
  END_VAR
                  {analysis -2} 
/// After leaving the state |STATE.DORMANT| the ``SampleAction`` is running one time then the state |STATE.STARTING| is reached.
/// If there is a ``iErrorID`` ≠  0 (Zero) the state |STATE.CLEANING| is reached instead.
///
/// .. note::
///
///    If this method will not provide any implementation, please remove it!

                
END_METHOD

METHOD StartAction
  VAR_OUTPUT
    xComplete : BOOL := TRUE;
    iErrorID : INT := 0;
  END_VAR
                  {analysis -2} 
/// The ``StartAction`` is running until either the output ``xComplete`` is ``TRUE`` or ``iErrorID`` ≠ 0 (Zero).
/// If ``xComplete`` is ``TRUE`` the state |STATE.EXECUTING| is reached.
/// If there is a ``iErrorID`` ≠  0 (Zero) the state |STATE.CLEANING| is reached.
///
/// .. note::
///
///    To sample the inputs in the first invocation of a function block the method SampleAction is the solution of choice.
///    See: |ISampleActionProvider.SampleAction|
///
/// .. note::
///
///    If this method will not provide any implementation, please remove it!

                
END_METHOD
END_FUNCTION_BLOCK

(* {attribute 'hide_all_locals'} {attribute 'conditionalshow_all_locals' := 'SomeText'} {attribute 'conditionalshow_all_locals'} {attribute 'conditionalshow' := 'SomeText'} {attribute 'conditionalshow'} {attribute 'hide'} *)
FUNCTION_BLOCK ETrigTo_Temp EXTENDS CBML.ETrigTo
  VAR_OUTPUT
    eErrorID : ERROR;
  END_VAR

            SUPER^();
IF _Model.iErrorID = CBML.ERROR.TIME_OUT THEN
	eErrorID := ERROR.TIME_OUT;
ELSE
	eErrorID := _Model.iErrorID;
END_IF

          

METHOD CleanupAction
  VAR_INPUT
    xAbortProposed : BOOL;
    iErrorIDProposed : INT;
  END_VAR
  VAR_OUTPUT
    xComplete : BOOL := TRUE;
    xAbort : BOOL := xAbortProposed;
    iErrorID : INT := iErrorIDProposed;
  END_VAR
                  {analysis -2} 
/// ``CleanupAction`` is running until one of the following events occurs:
/// When ``xComplete`` is ``TRUE`` the state |STATE.DONE| is reached.
/// When ``xAbort`` is ``TRUE`` the state |STATE.ABORTED| is reached.
/// When ``iErrorID`` ≠ 0 (Zero) the state |STATE.ERROR| is reached.
///
/// | After a *Ready Condition* as input (``iErrorIDProposed`` = 0 and ``xAbortProposed`` = ``FALSE``), only the output states
/// | `DONE` (``xComplete`` is ``TRUE``) or `ERROR` (``iErrorID`` ≠ 0) are possible.
///
/// | After a *Error Condition* as input (``iErrorIDProposed`` ≠ 0), only the output state
/// | `ERROR` (``iErrorID`` ≠ 0) is possible.
///
/// | After a *Abort Condition* as Input (``xAbortProposed`` = ``TRUE``), only the output states
/// | `ABORTED` (``xAbort`` is ``TRUE``) or `ERROR` (``iErrorID`` ≠ 0) are possible.
///
/// .. admonition:: Example
///
///     .. code-block:: codesys
///     
///         (* common cleanup -- first steps *) 
///         
///         IF xComplete THEN
///             IF xAbortProposed THEN
///                 (* abort condition -- abort specific cleanup *)
///                 xAbort := TRUE;
///                 xComplete := FALSE;
///             ELSIF iErrorIDProposed <> 0 THEN
///                 (* error condition -- error specific cleanup *)
///                 iErrorID := SEL(xComplete, 0, iErrorIDProposed);
///                 xComplete := FALSE;
///             ELSE
///                 (* ready condition -- done specific cleanup*)
///             END_IF
///         END_IF
///
///         (* common cleanup -- last steps *) 
///
/// .. note::
///
///    If this method will not provide any implementation, please remove it!

                
END_METHOD

METHOD CyclicAction
  VAR_INPUT
    itfTimingController : CBML.ITimingController;
  END_VAR
  VAR_OUTPUT
    xComplete : BOOL := TRUE;
    iErrorID : INT := 0;
  END_VAR
                  {analysis -2} 
/// The CyclicAction is running until either ``xComplete`` is ``TRUE`` or ``iErrorID`` ≠  0 (Zero).
/// If ``xComplete`` is ``TRUE`` or ``iErrorID`` ≠  0 (Zero) the state |STATE.CLEANING| is reached.
/// With ``itfTimingController`` ≠  0 (Zero) it is possible to check the current invocation time (see: |ITimingController.ControllerCheckTiming|).
/// Function blocks with a ``udiTimeLimit`` input variable (see: |IETrigTl|, |IETrigATl|, |IETrigTlTo|, |IETrigATlTo|, |ILConTl|, |ILConTlTo|, |ILConTlC|)
/// should be implement in such a way that the current invocation is exited when the consumed time for this invocation has exceeded the settings from udiTimeLimit.
///
/// .. admonition:: Example
///
///     .. code-block:: codesys
///     
///         REPEAT
///             // working to reach the ready condition
///             // ⇒ xComplete := TRUE
///             // if the maximum invocation time is reached
///             // ⇒ xTimeLimit := TRUE
///             // if the maximum operating time is reached
///             // ⇒ xTimeOut := TRUE
///             // if an error condition is reached
///             // ⇒ set iErrorID to a value other than 0 (Zero)
///             itfTimingController.ControllerCheckTiming(
///                 xTimeOut=>xTimeOut,
///                 xTimeLimit=>xTimeLimit
///             );
///         
///             xComplete := TRUE;
///             iErrorID := ERROR.NO_ERROR;
///     
///         UNTIL xComplete OR
///               xTimeOut OR xTimeLimit OR
///               iErrorID <> ERROR.NO_ERROR
///         END_REPEAT
///
/// .. note::
///
///    If this method will not provide any implementation, please remove it!

                
END_METHOD

METHOD ExitAction
  VAR_INPUT
    xAfterCleanup : BOOL;
    xInCopyCode : BOOL;
  END_VAR
                  {analysis -2} 
/// This method is intended for releasing external resources (like RTS handles).
/// Do not call other internal function block instances in the context of this method.
/// Call only external functions defined inside the RTS.
/// For cleaning up other resources then external ones, please use the ``CleanupAction``.
/// This method should be callable in the context of ``FB_EXIT`` for example
/// before downloading a new application or before reseting an application.
///
/// .. note::
///
///    If this method will not provide any implementation, please remove it!

                
END_METHOD

METHOD ResetAction
  VAR_OUTPUT
    xComplete : BOOL := TRUE;
  END_VAR
                  {analysis -2} 
/// The ``ResetAction`` is running until the output ``xComplete`` is ``TRUE``.
/// If ``xComplete`` is ``TRUE`` the state |STATE.DORMANT| is reached.
///
/// .. note::
///
///    If this method will not provide any implementation, please remove it!

                
END_METHOD

METHOD SampleAction
  VAR_OUTPUT
    iErrorID : INT := 0;
  END_VAR
                  {analysis -2} 
/// After leaving the state |STATE.DORMANT| the ``SampleAction`` is running one time then the state |STATE.STARTING| is reached.
/// If there is a ``iErrorID`` ≠  0 (Zero) the state |STATE.CLEANING| is reached instead.
///
/// .. note::
///
///    If this method will not provide any implementation, please remove it!

                
END_METHOD

METHOD StartAction
  VAR_OUTPUT
    xComplete : BOOL := TRUE;
    iErrorID : INT := 0;
  END_VAR
                  {analysis -2} 
/// The ``StartAction`` is running until either the output ``xComplete`` is ``TRUE`` or ``iErrorID`` ≠ 0 (Zero).
/// If ``xComplete`` is ``TRUE`` the state |STATE.EXECUTING| is reached.
/// If there is a ``iErrorID`` ≠  0 (Zero) the state |STATE.CLEANING| is reached.
///
/// .. note::
///
///    To sample the inputs in the first invocation of a function block the method SampleAction is the solution of choice.
///    See: |ISampleActionProvider.SampleAction|
///
/// .. note::
///
///    If this method will not provide any implementation, please remove it!

                
END_METHOD
END_FUNCTION_BLOCK

(* {attribute 'hide_all_locals'} {attribute 'conditionalshow_all_locals' := 'SomeText'} {attribute 'conditionalshow_all_locals'} {attribute 'conditionalshow' := 'SomeText'} {attribute 'conditionalshow'} {attribute 'hide'} *)
FUNCTION_BLOCK LCon_Temp EXTENDS CBML.LCon
  VAR_OUTPUT
    eErrorID : ERROR;
  END_VAR

            SUPER^();
eErrorID := _Model.iErrorID;


          

METHOD CleanupAction
  VAR_INPUT
    xAbortProposed : BOOL;
    iErrorIDProposed : INT;
  END_VAR
  VAR_OUTPUT
    xComplete : BOOL := TRUE;
    xAbort : BOOL := xAbortProposed;
    iErrorID : INT := iErrorIDProposed;
  END_VAR
                  {analysis -2} 
/// ``CleanupAction`` is running until one of the following events occurs:
/// When ``xComplete`` is ``TRUE`` the state |STATE.DONE| is reached.
/// When ``xAbort`` is ``TRUE`` the state |STATE.ABORTED| is reached.
/// When ``iErrorID`` ≠ 0 (Zero) the state |STATE.ERROR| is reached.
///
/// | After a *Ready Condition* as input (``iErrorIDProposed`` = 0 and ``xAbortProposed`` = ``FALSE``), only the output states
/// | `DONE` (``xComplete`` is ``TRUE``) or `ERROR` (``iErrorID`` ≠ 0) are possible.
///
/// | After a *Error Condition* as input (``iErrorIDProposed`` ≠ 0), only the output state
/// | `ERROR` (``iErrorID`` ≠ 0) is possible.
///
/// | After a *Abort Condition* as Input (``xAbortProposed`` = ``TRUE``), only the output states
/// | `ABORTED` (``xAbort`` is ``TRUE``) or `ERROR` (``iErrorID`` ≠ 0) are possible.
///
/// .. admonition:: Example
///
///     .. code-block:: codesys
///     
///         (* common cleanup -- first steps *) 
///         
///         IF xComplete THEN
///             IF xAbortProposed THEN
///                 (* abort condition -- abort specific cleanup *)
///                 xAbort := TRUE;
///                 xComplete := FALSE;
///             ELSIF iErrorIDProposed <> 0 THEN
///                 (* error condition -- error specific cleanup *)
///                 iErrorID := SEL(xComplete, 0, iErrorIDProposed);
///                 xComplete := FALSE;
///             ELSE
///                 (* ready condition -- done specific cleanup*)
///             END_IF
///         END_IF
///
///         (* common cleanup -- last steps *) 
///
/// .. note::
///
///    If this method will not provide any implementation, please remove it!

                
END_METHOD

METHOD CyclicAction
  VAR_INPUT
    itfTimingController : CBML.ITimingController;
  END_VAR
  VAR_OUTPUT
    xComplete : BOOL := TRUE;
    iErrorID : INT := 0;
  END_VAR
                  {analysis -2} 
/// The CyclicAction is running until either ``xComplete`` is ``TRUE`` or ``iErrorID`` ≠  0 (Zero).
/// If ``xComplete`` is ``TRUE`` or ``iErrorID`` ≠  0 (Zero) the state |STATE.CLEANING| is reached.
/// With ``itfTimingController`` ≠  0 (Zero) it is possible to check the current invocation time (see: |ITimingController.ControllerCheckTiming|).
/// Function blocks with a ``udiTimeLimit`` input variable (see: |IETrigTl|, |IETrigATl|, |IETrigTlTo|, |IETrigATlTo|, |ILConTl|, |ILConTlTo|, |ILConTlC|)
/// should be implement in such a way that the current invocation is exited when the consumed time for this invocation has exceeded the settings from udiTimeLimit.
///
/// .. admonition:: Example
///
///     .. code-block:: codesys
///     
///         REPEAT
///             // working to reach the ready condition
///             // ⇒ xComplete := TRUE
///             // if the maximum invocation time is reached
///             // ⇒ xTimeLimit := TRUE
///             // if the maximum operating time is reached
///             // ⇒ xTimeOut := TRUE
///             // if an error condition is reached
///             // ⇒ set iErrorID to a value other than 0 (Zero)
///             itfTimingController.ControllerCheckTiming(
///                 xTimeOut=>xTimeOut,
///                 xTimeLimit=>xTimeLimit
///             );
///         
///             xComplete := TRUE;
///             iErrorID := ERROR.NO_ERROR;
///     
///         UNTIL xComplete OR
///               xTimeOut OR xTimeLimit OR
///               iErrorID <> ERROR.NO_ERROR
///         END_REPEAT
///
/// .. note::
///
///    If this method will not provide any implementation, please remove it!

                
END_METHOD

METHOD ExitAction
  VAR_INPUT
    xAfterCleanup : BOOL;
    xInCopyCode : BOOL;
  END_VAR
                  {analysis -2} 
/// This method is intended for releasing external resources (like RTS handles).
/// Do not call other internal function block instances in the context of this method.
/// Call only external functions defined inside the RTS.
/// For cleaning up other resources then external ones, please use the ``CleanupAction``.
/// This method should be callable in the context of ``FB_EXIT`` for example
/// before downloading a new application or before reseting an application.
///
/// .. note::
///
///    If this method will not provide any implementation, please remove it!

                
END_METHOD

METHOD ResetAction
  VAR_OUTPUT
    xComplete : BOOL := TRUE;
  END_VAR
                  {analysis -2} 
/// The ``ResetAction`` is running until the output ``xComplete`` is ``TRUE``.
/// If ``xComplete`` is ``TRUE`` the state |STATE.DORMANT| is reached.
///
/// .. note::
///
///    If this method will not provide any implementation, please remove it!

                
END_METHOD

METHOD StartAction
  VAR_OUTPUT
    xComplete : BOOL := TRUE;
    iErrorID : INT := 0;
  END_VAR
                  {analysis -2} 
/// The ``StartAction`` is running until either the output ``xComplete`` is ``TRUE`` or ``iErrorID`` ≠ 0 (Zero).
/// If ``xComplete`` is ``TRUE`` the state |STATE.EXECUTING| is reached.
/// If there is a ``iErrorID`` ≠  0 (Zero) the state |STATE.CLEANING| is reached.
///
/// .. note::
///
///    To sample the inputs in the first invocation of a function block the method SampleAction is the solution of choice.
///    See: |ISampleActionProvider.SampleAction|
///
/// .. note::
///
///    If this method will not provide any implementation, please remove it!

                
END_METHOD
END_FUNCTION_BLOCK

(* {attribute 'hide_all_locals'} {attribute 'conditionalshow_all_locals' := 'SomeText'} {attribute 'conditionalshow_all_locals'} {attribute 'conditionalshow' := 'SomeText'} {attribute 'conditionalshow'} {attribute 'hide'} *)
FUNCTION_BLOCK LConC_Temp EXTENDS CBML.LConC
  VAR_OUTPUT
    eErrorID : ERROR;
  END_VAR

            SUPER^();
eErrorID := _Model.iErrorID;


          

METHOD CleanupAction
  VAR_INPUT
    xAbortProposed : BOOL;
    iErrorIDProposed : INT;
  END_VAR
  VAR_OUTPUT
    xComplete : BOOL := TRUE;
    xAbort : BOOL := xAbortProposed;
    iErrorID : INT := iErrorIDProposed;
  END_VAR
                  {analysis -2} 
/// ``CleanupAction`` is running until one of the following events occurs:
/// When ``xComplete`` is ``TRUE`` the state |STATE.DONE| is reached.
/// When ``xAbort`` is ``TRUE`` the state |STATE.ABORTED| is reached.
/// When ``iErrorID`` ≠ 0 (Zero) the state |STATE.ERROR| is reached.
///
/// | After a *Ready Condition* as input (``iErrorIDProposed`` = 0 and ``xAbortProposed`` = ``FALSE``), only the output states
/// | `DONE` (``xComplete`` is ``TRUE``) or `ERROR` (``iErrorID`` ≠ 0) are possible.
///
/// | After a *Error Condition* as input (``iErrorIDProposed`` ≠ 0), only the output state
/// | `ERROR` (``iErrorID`` ≠ 0) is possible.
///
/// | After a *Abort Condition* as Input (``xAbortProposed`` = ``TRUE``), only the output states
/// | `ABORTED` (``xAbort`` is ``TRUE``) or `ERROR` (``iErrorID`` ≠ 0) are possible.
///
/// .. admonition:: Example
///
///     .. code-block:: codesys
///     
///         (* common cleanup -- first steps *) 
///         
///         IF xComplete THEN
///             IF xAbortProposed THEN
///                 (* abort condition -- abort specific cleanup *)
///                 xAbort := TRUE;
///                 xComplete := FALSE;
///             ELSIF iErrorIDProposed <> 0 THEN
///                 (* error condition -- error specific cleanup *)
///                 iErrorID := SEL(xComplete, 0, iErrorIDProposed);
///                 xComplete := FALSE;
///             ELSE
///                 (* ready condition -- done specific cleanup*)
///             END_IF
///         END_IF
///
///         (* common cleanup -- last steps *) 
///
/// .. note::
///
///    If this method will not provide any implementation, please remove it!

                
END_METHOD

METHOD CyclicAction
  VAR_INPUT
    itfTimingController : CBML.ITimingController;
  END_VAR
  VAR_OUTPUT
    xComplete : BOOL := TRUE;
    iErrorID : INT := 0;
  END_VAR
                  {analysis -2} 
/// The CyclicAction is running until either ``xComplete`` is ``TRUE`` or ``iErrorID`` ≠  0 (Zero).
/// If ``xComplete`` is ``TRUE`` or ``iErrorID`` ≠  0 (Zero) the state |STATE.CLEANING| is reached.
/// With ``itfTimingController`` ≠  0 (Zero) it is possible to check the current invocation time (see: |ITimingController.ControllerCheckTiming|).
/// Function blocks with a ``udiTimeLimit`` input variable (see: |IETrigTl|, |IETrigATl|, |IETrigTlTo|, |IETrigATlTo|, |ILConTl|, |ILConTlTo|, |ILConTlC|)
/// should be implement in such a way that the current invocation is exited when the consumed time for this invocation has exceeded the settings from udiTimeLimit.
///
/// .. admonition:: Example
///
///     .. code-block:: codesys
///     
///         REPEAT
///             // working to reach the ready condition
///             // ⇒ xComplete := TRUE
///             // if the maximum invocation time is reached
///             // ⇒ xTimeLimit := TRUE
///             // if the maximum operating time is reached
///             // ⇒ xTimeOut := TRUE
///             // if an error condition is reached
///             // ⇒ set iErrorID to a value other than 0 (Zero)
///             itfTimingController.ControllerCheckTiming(
///                 xTimeOut=>xTimeOut,
///                 xTimeLimit=>xTimeLimit
///             );
///         
///             xComplete := TRUE;
///             iErrorID := ERROR.NO_ERROR;
///     
///         UNTIL xComplete OR
///               xTimeOut OR xTimeLimit OR
///               iErrorID <> ERROR.NO_ERROR
///         END_REPEAT
///
/// .. note::
///
///    If this method will not provide any implementation, please remove it!

                
END_METHOD

METHOD ExitAction
  VAR_INPUT
    xAfterCleanup : BOOL;
    xInCopyCode : BOOL;
  END_VAR
                  {analysis -2} 
/// This method is intended for releasing external resources (like RTS handles).
/// Do not call other internal function block instances in the context of this method.
/// Call only external functions defined inside the RTS.
/// For cleaning up other resources then external ones, please use the ``CleanupAction``.
/// This method should be callable in the context of ``FB_EXIT`` for example
/// before downloading a new application or before reseting an application.
///
/// .. note::
///
///    If this method will not provide any implementation, please remove it!

                
END_METHOD

METHOD ResetAction
  VAR_OUTPUT
    xComplete : BOOL := TRUE;
  END_VAR
                  {analysis -2} 
/// The ``ResetAction`` is running until the output ``xComplete`` is ``TRUE``.
/// If ``xComplete`` is ``TRUE`` the state |STATE.DORMANT| is reached.
///
/// .. note::
///
///    If this method will not provide any implementation, please remove it!

                
END_METHOD

METHOD StartAction
  VAR_OUTPUT
    xComplete : BOOL := TRUE;
    iErrorID : INT := 0;
  END_VAR
                  {analysis -2} 
/// The ``StartAction`` is running until either the output ``xComplete`` is ``TRUE`` or ``iErrorID`` ≠ 0 (Zero).
/// If ``xComplete`` is ``TRUE`` the state |STATE.EXECUTING| is reached.
/// If there is a ``iErrorID`` ≠  0 (Zero) the state |STATE.CLEANING| is reached.
///
/// .. note::
///
///    To sample the inputs in the first invocation of a function block the method SampleAction is the solution of choice.
///    See: |ISampleActionProvider.SampleAction|
///
/// .. note::
///
///    If this method will not provide any implementation, please remove it!

                
END_METHOD
END_FUNCTION_BLOCK

(* {attribute 'hide_all_locals'} {attribute 'conditionalshow_all_locals' := 'SomeText'} {attribute 'conditionalshow_all_locals'} {attribute 'conditionalshow' := 'SomeText'} {attribute 'conditionalshow'} {attribute 'hide'} *)
FUNCTION_BLOCK LConTl_Temp EXTENDS CBML.LConTl
  VAR_OUTPUT
    eErrorID : ERROR;
  END_VAR

            SUPER^();
eErrorID := _Model.iErrorID;


          

METHOD CleanupAction
  VAR_INPUT
    xAbortProposed : BOOL;
    iErrorIDProposed : INT;
  END_VAR
  VAR_OUTPUT
    xComplete : BOOL := TRUE;
    xAbort : BOOL := xAbortProposed;
    iErrorID : INT := iErrorIDProposed;
  END_VAR
                  {analysis -2} 
/// ``CleanupAction`` is running until one of the following events occurs:
/// When ``xComplete`` is ``TRUE`` the state |STATE.DONE| is reached.
/// When ``xAbort`` is ``TRUE`` the state |STATE.ABORTED| is reached.
/// When ``iErrorID`` ≠ 0 (Zero) the state |STATE.ERROR| is reached.
///
/// | After a *Ready Condition* as input (``iErrorIDProposed`` = 0 and ``xAbortProposed`` = ``FALSE``), only the output states
/// | `DONE` (``xComplete`` is ``TRUE``) or `ERROR` (``iErrorID`` ≠ 0) are possible.
///
/// | After a *Error Condition* as input (``iErrorIDProposed`` ≠ 0), only the output state
/// | `ERROR` (``iErrorID`` ≠ 0) is possible.
///
/// | After a *Abort Condition* as Input (``xAbortProposed`` = ``TRUE``), only the output states
/// | `ABORTED` (``xAbort`` is ``TRUE``) or `ERROR` (``iErrorID`` ≠ 0) are possible.
///
/// .. admonition:: Example
///
///     .. code-block:: codesys
///     
///         (* common cleanup -- first steps *) 
///         
///         IF xComplete THEN
///             IF xAbortProposed THEN
///                 (* abort condition -- abort specific cleanup *)
///                 xAbort := TRUE;
///                 xComplete := FALSE;
///             ELSIF iErrorIDProposed <> 0 THEN
///                 (* error condition -- error specific cleanup *)
///                 iErrorID := SEL(xComplete, 0, iErrorIDProposed);
///                 xComplete := FALSE;
///             ELSE
///                 (* ready condition -- done specific cleanup*)
///             END_IF
///         END_IF
///
///         (* common cleanup -- last steps *) 
///
/// .. note::
///
///    If this method will not provide any implementation, please remove it!

                
END_METHOD

METHOD CyclicAction
  VAR_INPUT
    itfTimingController : CBML.ITimingController;
  END_VAR
  VAR_OUTPUT
    xComplete : BOOL := TRUE;
    iErrorID : INT := 0;
  END_VAR
                  {analysis -2} 
/// The CyclicAction is running until either ``xComplete`` is ``TRUE`` or ``iErrorID`` ≠  0 (Zero).
/// If ``xComplete`` is ``TRUE`` or ``iErrorID`` ≠  0 (Zero) the state |STATE.CLEANING| is reached.
/// With ``itfTimingController`` ≠  0 (Zero) it is possible to check the current invocation time (see: |ITimingController.ControllerCheckTiming|).
/// Function blocks with a ``udiTimeLimit`` input variable (see: |IETrigTl|, |IETrigATl|, |IETrigTlTo|, |IETrigATlTo|, |ILConTl|, |ILConTlTo|, |ILConTlC|)
/// should be implement in such a way that the current invocation is exited when the consumed time for this invocation has exceeded the settings from udiTimeLimit.
///
/// .. admonition:: Example
///
///     .. code-block:: codesys
///     
///         REPEAT
///             // working to reach the ready condition
///             // ⇒ xComplete := TRUE
///             // if the maximum invocation time is reached
///             // ⇒ xTimeLimit := TRUE
///             // if the maximum operating time is reached
///             // ⇒ xTimeOut := TRUE
///             // if an error condition is reached
///             // ⇒ set iErrorID to a value other than 0 (Zero)
///             itfTimingController.ControllerCheckTiming(
///                 xTimeOut=>xTimeOut,
///                 xTimeLimit=>xTimeLimit
///             );
///         
///             xComplete := TRUE;
///             iErrorID := ERROR.NO_ERROR;
///     
///         UNTIL xComplete OR
///               xTimeOut OR xTimeLimit OR
///               iErrorID <> ERROR.NO_ERROR
///         END_REPEAT
///
/// .. note::
///
///    If this method will not provide any implementation, please remove it!

                
END_METHOD

METHOD ExitAction
  VAR_INPUT
    xAfterCleanup : BOOL;
    xInCopyCode : BOOL;
  END_VAR
                  {analysis -2} 
/// This method is intended for releasing external resources (like RTS handles).
/// Do not call other internal function block instances in the context of this method.
/// Call only external functions defined inside the RTS.
/// For cleaning up other resources then external ones, please use the ``CleanupAction``.
/// This method should be callable in the context of ``FB_EXIT`` for example
/// before downloading a new application or before reseting an application.
///
/// .. note::
///
///    If this method will not provide any implementation, please remove it!

                
END_METHOD

METHOD ResetAction
  VAR_OUTPUT
    xComplete : BOOL := TRUE;
  END_VAR
                  {analysis -2} 
/// The ``ResetAction`` is running until the output ``xComplete`` is ``TRUE``.
/// If ``xComplete`` is ``TRUE`` the state |STATE.DORMANT| is reached.
///
/// .. note::
///
///    If this method will not provide any implementation, please remove it!

                
END_METHOD

METHOD StartAction
  VAR_OUTPUT
    xComplete : BOOL := TRUE;
    iErrorID : INT := 0;
  END_VAR
                  {analysis -2} 
/// The ``StartAction`` is running until either the output ``xComplete`` is ``TRUE`` or ``iErrorID`` ≠ 0 (Zero).
/// If ``xComplete`` is ``TRUE`` the state |STATE.EXECUTING| is reached.
/// If there is a ``iErrorID`` ≠  0 (Zero) the state |STATE.CLEANING| is reached.
///
/// .. note::
///
///    To sample the inputs in the first invocation of a function block the method SampleAction is the solution of choice.
///    See: |ISampleActionProvider.SampleAction|
///
/// .. note::
///
///    If this method will not provide any implementation, please remove it!

                
END_METHOD
END_FUNCTION_BLOCK

(* {attribute 'hide_all_locals'} {attribute 'conditionalshow_all_locals' := 'SomeText'} {attribute 'conditionalshow_all_locals'} {attribute 'conditionalshow' := 'SomeText'} {attribute 'conditionalshow'} {attribute 'hide'} *)
FUNCTION_BLOCK LConTlC_Temp EXTENDS CBML.LConTlC
  VAR_OUTPUT
    eErrorID : ERROR;
  END_VAR

            SUPER^();
eErrorID := _Model.iErrorID;


          

METHOD CleanupAction
  VAR_INPUT
    xAbortProposed : BOOL;
    iErrorIDProposed : INT;
  END_VAR
  VAR_OUTPUT
    xComplete : BOOL := TRUE;
    xAbort : BOOL := xAbortProposed;
    iErrorID : INT := iErrorIDProposed;
  END_VAR
                  {analysis -2} 
/// ``CleanupAction`` is running until one of the following events occurs:
/// When ``xComplete`` is ``TRUE`` the state |STATE.DONE| is reached.
/// When ``xAbort`` is ``TRUE`` the state |STATE.ABORTED| is reached.
/// When ``iErrorID`` ≠ 0 (Zero) the state |STATE.ERROR| is reached.
///
/// | After a *Ready Condition* as input (``iErrorIDProposed`` = 0 and ``xAbortProposed`` = ``FALSE``), only the output states
/// | `DONE` (``xComplete`` is ``TRUE``) or `ERROR` (``iErrorID`` ≠ 0) are possible.
///
/// | After a *Error Condition* as input (``iErrorIDProposed`` ≠ 0), only the output state
/// | `ERROR` (``iErrorID`` ≠ 0) is possible.
///
/// | After a *Abort Condition* as Input (``xAbortProposed`` = ``TRUE``), only the output states
/// | `ABORTED` (``xAbort`` is ``TRUE``) or `ERROR` (``iErrorID`` ≠ 0) are possible.
///
/// .. admonition:: Example
///
///     .. code-block:: codesys
///     
///         (* common cleanup -- first steps *) 
///         
///         IF xComplete THEN
///             IF xAbortProposed THEN
///                 (* abort condition -- abort specific cleanup *)
///                 xAbort := TRUE;
///                 xComplete := FALSE;
///             ELSIF iErrorIDProposed <> 0 THEN
///                 (* error condition -- error specific cleanup *)
///                 iErrorID := SEL(xComplete, 0, iErrorIDProposed);
///                 xComplete := FALSE;
///             ELSE
///                 (* ready condition -- done specific cleanup*)
///             END_IF
///         END_IF
///
///         (* common cleanup -- last steps *) 
///
/// .. note::
///
///    If this method will not provide any implementation, please remove it!

                
END_METHOD

METHOD CyclicAction
  VAR_INPUT
    itfTimingController : CBML.ITimingController;
  END_VAR
  VAR_OUTPUT
    xComplete : BOOL := TRUE;
    iErrorID : INT := 0;
  END_VAR
                  {analysis -2} 
/// The CyclicAction is running until either ``xComplete`` is ``TRUE`` or ``iErrorID`` ≠  0 (Zero).
/// If ``xComplete`` is ``TRUE`` or ``iErrorID`` ≠  0 (Zero) the state |STATE.CLEANING| is reached.
/// With ``itfTimingController`` ≠  0 (Zero) it is possible to check the current invocation time (see: |ITimingController.ControllerCheckTiming|).
/// Function blocks with a ``udiTimeLimit`` input variable (see: |IETrigTl|, |IETrigATl|, |IETrigTlTo|, |IETrigATlTo|, |ILConTl|, |ILConTlTo|, |ILConTlC|)
/// should be implement in such a way that the current invocation is exited when the consumed time for this invocation has exceeded the settings from udiTimeLimit.
///
/// .. admonition:: Example
///
///     .. code-block:: codesys
///     
///         REPEAT
///             // working to reach the ready condition
///             // ⇒ xComplete := TRUE
///             // if the maximum invocation time is reached
///             // ⇒ xTimeLimit := TRUE
///             // if the maximum operating time is reached
///             // ⇒ xTimeOut := TRUE
///             // if an error condition is reached
///             // ⇒ set iErrorID to a value other than 0 (Zero)
///             itfTimingController.ControllerCheckTiming(
///                 xTimeOut=>xTimeOut,
///                 xTimeLimit=>xTimeLimit
///             );
///         
///             xComplete := TRUE;
///             iErrorID := ERROR.NO_ERROR;
///     
///         UNTIL xComplete OR
///               xTimeOut OR xTimeLimit OR
///               iErrorID <> ERROR.NO_ERROR
///         END_REPEAT
///
/// .. note::
///
///    If this method will not provide any implementation, please remove it!

                
END_METHOD

METHOD ExitAction
  VAR_INPUT
    xAfterCleanup : BOOL;
    xInCopyCode : BOOL;
  END_VAR
                  {analysis -2} 
/// This method is intended for releasing external resources (like RTS handles).
/// Do not call other internal function block instances in the context of this method.
/// Call only external functions defined inside the RTS.
/// For cleaning up other resources then external ones, please use the ``CleanupAction``.
/// This method should be callable in the context of ``FB_EXIT`` for example
/// before downloading a new application or before reseting an application.
///
/// .. note::
///
///    If this method will not provide any implementation, please remove it!

                
END_METHOD

METHOD ResetAction
  VAR_OUTPUT
    xComplete : BOOL := TRUE;
  END_VAR
                  {analysis -2} 
/// The ``ResetAction`` is running until the output ``xComplete`` is ``TRUE``.
/// If ``xComplete`` is ``TRUE`` the state |STATE.DORMANT| is reached.
///
/// .. note::
///
///    If this method will not provide any implementation, please remove it!

                
END_METHOD

METHOD StartAction
  VAR_OUTPUT
    xComplete : BOOL := TRUE;
    iErrorID : INT := 0;
  END_VAR
                  {analysis -2} 
/// The ``StartAction`` is running until either the output ``xComplete`` is ``TRUE`` or ``iErrorID`` ≠ 0 (Zero).
/// If ``xComplete`` is ``TRUE`` the state |STATE.EXECUTING| is reached.
/// If there is a ``iErrorID`` ≠  0 (Zero) the state |STATE.CLEANING| is reached.
///
/// .. note::
///
///    To sample the inputs in the first invocation of a function block the method SampleAction is the solution of choice.
///    See: |ISampleActionProvider.SampleAction|
///
/// .. note::
///
///    If this method will not provide any implementation, please remove it!

                
END_METHOD
END_FUNCTION_BLOCK

(* {attribute 'hide_all_locals'} {attribute 'conditionalshow_all_locals' := 'SomeText'} {attribute 'conditionalshow_all_locals'} {attribute 'conditionalshow' := 'SomeText'} {attribute 'conditionalshow'} {attribute 'hide'} *)
FUNCTION_BLOCK LConTlTo_Temp EXTENDS CBML.LConTlTo
  VAR_OUTPUT
    eErrorID : ERROR;
  END_VAR

            SUPER^();
IF _Model.iErrorID = CBML.ERROR.TIME_OUT THEN
	eErrorID := ERROR.TIME_OUT;
ELSE
	eErrorID := _Model.iErrorID;
END_IF

          

METHOD CleanupAction
  VAR_INPUT
    xAbortProposed : BOOL;
    iErrorIDProposed : INT;
  END_VAR
  VAR_OUTPUT
    xComplete : BOOL := TRUE;
    xAbort : BOOL := xAbortProposed;
    iErrorID : INT := iErrorIDProposed;
  END_VAR
                  {analysis -2} 
/// ``CleanupAction`` is running until one of the following events occurs:
/// When ``xComplete`` is ``TRUE`` the state |STATE.DONE| is reached.
/// When ``xAbort`` is ``TRUE`` the state |STATE.ABORTED| is reached.
/// When ``iErrorID`` ≠ 0 (Zero) the state |STATE.ERROR| is reached.
///
/// | After a *Ready Condition* as input (``iErrorIDProposed`` = 0 and ``xAbortProposed`` = ``FALSE``), only the output states
/// | `DONE` (``xComplete`` is ``TRUE``) or `ERROR` (``iErrorID`` ≠ 0) are possible.
///
/// | After a *Error Condition* as input (``iErrorIDProposed`` ≠ 0), only the output state
/// | `ERROR` (``iErrorID`` ≠ 0) is possible.
///
/// | After a *Abort Condition* as Input (``xAbortProposed`` = ``TRUE``), only the output states
/// | `ABORTED` (``xAbort`` is ``TRUE``) or `ERROR` (``iErrorID`` ≠ 0) are possible.
///
/// .. admonition:: Example
///
///     .. code-block:: codesys
///     
///         (* common cleanup -- first steps *) 
///         
///         IF xComplete THEN
///             IF xAbortProposed THEN
///                 (* abort condition -- abort specific cleanup *)
///                 xAbort := TRUE;
///                 xComplete := FALSE;
///             ELSIF iErrorIDProposed <> 0 THEN
///                 (* error condition -- error specific cleanup *)
///                 iErrorID := SEL(xComplete, 0, iErrorIDProposed);
///                 xComplete := FALSE;
///             ELSE
///                 (* ready condition -- done specific cleanup*)
///             END_IF
///         END_IF
///
///         (* common cleanup -- last steps *) 
///
/// .. note::
///
///    If this method will not provide any implementation, please remove it!

                
END_METHOD

METHOD CyclicAction
  VAR_INPUT
    itfTimingController : CBML.ITimingController;
  END_VAR
  VAR_OUTPUT
    xComplete : BOOL := TRUE;
    iErrorID : INT := 0;
  END_VAR
                  {analysis -2} 
/// The CyclicAction is running until either ``xComplete`` is ``TRUE`` or ``iErrorID`` ≠  0 (Zero).
/// If ``xComplete`` is ``TRUE`` or ``iErrorID`` ≠  0 (Zero) the state |STATE.CLEANING| is reached.
/// With ``itfTimingController`` ≠  0 (Zero) it is possible to check the current invocation time (see: |ITimingController.ControllerCheckTiming|).
/// Function blocks with a ``udiTimeLimit`` input variable (see: |IETrigTl|, |IETrigATl|, |IETrigTlTo|, |IETrigATlTo|, |ILConTl|, |ILConTlTo|, |ILConTlC|)
/// should be implement in such a way that the current invocation is exited when the consumed time for this invocation has exceeded the settings from udiTimeLimit.
///
/// .. admonition:: Example
///
///     .. code-block:: codesys
///     
///         REPEAT
///             // working to reach the ready condition
///             // ⇒ xComplete := TRUE
///             // if the maximum invocation time is reached
///             // ⇒ xTimeLimit := TRUE
///             // if the maximum operating time is reached
///             // ⇒ xTimeOut := TRUE
///             // if an error condition is reached
///             // ⇒ set iErrorID to a value other than 0 (Zero)
///             itfTimingController.ControllerCheckTiming(
///                 xTimeOut=>xTimeOut,
///                 xTimeLimit=>xTimeLimit
///             );
///         
///             xComplete := TRUE;
///             iErrorID := ERROR.NO_ERROR;
///     
///         UNTIL xComplete OR
///               xTimeOut OR xTimeLimit OR
///               iErrorID <> ERROR.NO_ERROR
///         END_REPEAT
///
/// .. note::
///
///    If this method will not provide any implementation, please remove it!

                
END_METHOD

METHOD ExitAction
  VAR_INPUT
    xAfterCleanup : BOOL;
    xInCopyCode : BOOL;
  END_VAR
                  {analysis -2} 
/// This method is intended for releasing external resources (like RTS handles).
/// Do not call other internal function block instances in the context of this method.
/// Call only external functions defined inside the RTS.
/// For cleaning up other resources then external ones, please use the ``CleanupAction``.
/// This method should be callable in the context of ``FB_EXIT`` for example
/// before downloading a new application or before reseting an application.
///
/// .. note::
///
///    If this method will not provide any implementation, please remove it!

                
END_METHOD

METHOD ResetAction
  VAR_OUTPUT
    xComplete : BOOL := TRUE;
  END_VAR
                  {analysis -2} 
/// The ``ResetAction`` is running until the output ``xComplete`` is ``TRUE``.
/// If ``xComplete`` is ``TRUE`` the state |STATE.DORMANT| is reached.
///
/// .. note::
///
///    If this method will not provide any implementation, please remove it!

                
END_METHOD

METHOD StartAction
  VAR_OUTPUT
    xComplete : BOOL := TRUE;
    iErrorID : INT := 0;
  END_VAR
                  {analysis -2} 
/// The ``StartAction`` is running until either the output ``xComplete`` is ``TRUE`` or ``iErrorID`` ≠ 0 (Zero).
/// If ``xComplete`` is ``TRUE`` the state |STATE.EXECUTING| is reached.
/// If there is a ``iErrorID`` ≠  0 (Zero) the state |STATE.CLEANING| is reached.
///
/// .. note::
///
///    To sample the inputs in the first invocation of a function block the method SampleAction is the solution of choice.
///    See: |ISampleActionProvider.SampleAction|
///
/// .. note::
///
///    If this method will not provide any implementation, please remove it!

                
END_METHOD
END_FUNCTION_BLOCK

(* {attribute 'hide_all_locals'} {attribute 'conditionalshow_all_locals' := 'SomeText'} {attribute 'conditionalshow_all_locals'} {attribute 'conditionalshow' := 'SomeText'} {attribute 'conditionalshow'} {attribute 'hide'} *)
FUNCTION_BLOCK LConTo_Temp EXTENDS CBML.LConTo
  VAR_OUTPUT
    eErrorID : ERROR;
  END_VAR

            SUPER^();
IF _Model.iErrorID = CBML.ERROR.TIME_OUT THEN
	eErrorID := ERROR.TIME_OUT;
ELSE
	eErrorID := _Model.iErrorID;
END_IF

          

METHOD CleanupAction
  VAR_INPUT
    xAbortProposed : BOOL;
    iErrorIDProposed : INT;
  END_VAR
  VAR_OUTPUT
    xComplete : BOOL := TRUE;
    xAbort : BOOL := xAbortProposed;
    iErrorID : INT := iErrorIDProposed;
  END_VAR
                  {analysis -2} 
/// ``CleanupAction`` is running until one of the following events occurs:
/// When ``xComplete`` is ``TRUE`` the state |STATE.DONE| is reached.
/// When ``xAbort`` is ``TRUE`` the state |STATE.ABORTED| is reached.
/// When ``iErrorID`` ≠ 0 (Zero) the state |STATE.ERROR| is reached.
///
/// | After a *Ready Condition* as input (``iErrorIDProposed`` = 0 and ``xAbortProposed`` = ``FALSE``), only the output states
/// | `DONE` (``xComplete`` is ``TRUE``) or `ERROR` (``iErrorID`` ≠ 0) are possible.
///
/// | After a *Error Condition* as input (``iErrorIDProposed`` ≠ 0), only the output state
/// | `ERROR` (``iErrorID`` ≠ 0) is possible.
///
/// | After a *Abort Condition* as Input (``xAbortProposed`` = ``TRUE``), only the output states
/// | `ABORTED` (``xAbort`` is ``TRUE``) or `ERROR` (``iErrorID`` ≠ 0) are possible.
///
/// .. admonition:: Example
///
///     .. code-block:: codesys
///     
///         (* common cleanup -- first steps *) 
///         
///         IF xComplete THEN
///             IF xAbortProposed THEN
///                 (* abort condition -- abort specific cleanup *)
///                 xAbort := TRUE;
///                 xComplete := FALSE;
///             ELSIF iErrorIDProposed <> 0 THEN
///                 (* error condition -- error specific cleanup *)
///                 iErrorID := SEL(xComplete, 0, iErrorIDProposed);
///                 xComplete := FALSE;
///             ELSE
///                 (* ready condition -- done specific cleanup*)
///             END_IF
///         END_IF
///
///         (* common cleanup -- last steps *) 
///
/// .. note::
///
///    If this method will not provide any implementation, please remove it!

                
END_METHOD

METHOD CyclicAction
  VAR_INPUT
    itfTimingController : CBML.ITimingController;
  END_VAR
  VAR_OUTPUT
    xComplete : BOOL := TRUE;
    iErrorID : INT := 0;
  END_VAR
                  {analysis -2} 
/// The CyclicAction is running until either ``xComplete`` is ``TRUE`` or ``iErrorID`` ≠  0 (Zero).
/// If ``xComplete`` is ``TRUE`` or ``iErrorID`` ≠  0 (Zero) the state |STATE.CLEANING| is reached.
/// With ``itfTimingController`` ≠  0 (Zero) it is possible to check the current invocation time (see: |ITimingController.ControllerCheckTiming|).
/// Function blocks with a ``udiTimeLimit`` input variable (see: |IETrigTl|, |IETrigATl|, |IETrigTlTo|, |IETrigATlTo|, |ILConTl|, |ILConTlTo|, |ILConTlC|)
/// should be implement in such a way that the current invocation is exited when the consumed time for this invocation has exceeded the settings from udiTimeLimit.
///
/// .. admonition:: Example
///
///     .. code-block:: codesys
///     
///         REPEAT
///             // working to reach the ready condition
///             // ⇒ xComplete := TRUE
///             // if the maximum invocation time is reached
///             // ⇒ xTimeLimit := TRUE
///             // if the maximum operating time is reached
///             // ⇒ xTimeOut := TRUE
///             // if an error condition is reached
///             // ⇒ set iErrorID to a value other than 0 (Zero)
///             itfTimingController.ControllerCheckTiming(
///                 xTimeOut=>xTimeOut,
///                 xTimeLimit=>xTimeLimit
///             );
///         
///             xComplete := TRUE;
///             iErrorID := ERROR.NO_ERROR;
///     
///         UNTIL xComplete OR
///               xTimeOut OR xTimeLimit OR
///               iErrorID <> ERROR.NO_ERROR
///         END_REPEAT
///
/// .. note::
///
///    If this method will not provide any implementation, please remove it!

                
END_METHOD

METHOD ExitAction
  VAR_INPUT
    xAfterCleanup : BOOL;
    xInCopyCode : BOOL;
  END_VAR
                  {analysis -2} 
/// This method is intended for releasing external resources (like RTS handles).
/// Do not call other internal function block instances in the context of this method.
/// Call only external functions defined inside the RTS.
/// For cleaning up other resources then external ones, please use the ``CleanupAction``.
/// This method should be callable in the context of ``FB_EXIT`` for example
/// before downloading a new application or before reseting an application.
///
/// .. note::
///
///    If this method will not provide any implementation, please remove it!

                
END_METHOD

METHOD ResetAction
  VAR_OUTPUT
    xComplete : BOOL := TRUE;
  END_VAR
                  {analysis -2} 
/// The ``ResetAction`` is running until the output ``xComplete`` is ``TRUE``.
/// If ``xComplete`` is ``TRUE`` the state |STATE.DORMANT| is reached.
///
/// .. note::
///
///    If this method will not provide any implementation, please remove it!

                
END_METHOD

METHOD StartAction
  VAR_OUTPUT
    xComplete : BOOL := TRUE;
    iErrorID : INT := 0;
  END_VAR
                  {analysis -2} 
/// The ``StartAction`` is running until either the output ``xComplete`` is ``TRUE`` or ``iErrorID`` ≠ 0 (Zero).
/// If ``xComplete`` is ``TRUE`` the state |STATE.EXECUTING| is reached.
/// If there is a ``iErrorID`` ≠  0 (Zero) the state |STATE.CLEANING| is reached.
///
/// .. note::
///
///    To sample the inputs in the first invocation of a function block the method SampleAction is the solution of choice.
///    See: |ISampleActionProvider.SampleAction|
///
/// .. note::
///
///    If this method will not provide any implementation, please remove it!

                
END_METHOD
END_FUNCTION_BLOCK

(* This is a container to carry init data from the Create methode of the factory to the prvInstInit methode of the new generated function block instance {attribute 'hide_all_locals'} {attribute 'conditionalshow_all_locals' := 'SomeText'} {attribute 'conditionalshow_all_locals'} {attribute 'conditionalshow' := 'SomeText'} {attribute 'conditionalshow'} {attribute 'hide'} *)
{attribute 'enable_dynamic_creation'}
FUNCTION_BLOCK CustomData EXTENDS FBF.InstanceData

            (* !! Do not add any executable code here !! *)
SUPER^();
          
END_FUNCTION_BLOCK

(* {attribute 'hide_all_locals'} {attribute 'conditionalshow_all_locals' := 'SomeText'} {attribute 'conditionalshow_all_locals'} {attribute 'conditionalshow' := 'SomeText'} {attribute 'conditionalshow'} {attribute 'hide'} *)
{attribute 'enable_dynamic_creation'}
FUNCTION_BLOCK CustomFB EXTENDS FBF.InstanceBase

            SUPER^();

          

(* This methode is called from the factory to give a chance to initialize the new fb instance with the content of itfData {attribute 'hide_all_locals'} {attribute 'conditionalshow_all_locals' := 'SomeText'} {attribute 'conditionalshow_all_locals'} {attribute 'conditionalshow' := 'SomeText'} {attribute 'conditionalshow'} {attribute 'hide'} *)
METHOD prvInstInit : FBF.ERROR
  VAR_INPUT
    itfData : FBF.IData;
  END_VAR
  VAR
    pData : POINTER TO CustomData;
    xOk : BOOL;
  END_VAR
                  SUPER^.prvInstInit(itfData);
xOk := __QUERYPOINTER(itfData, pData);
IF xOk THEN
	(* THIS^.iLocalVar := pData^.iInitValue *);
END_IF

                
END_METHOD
END_FUNCTION_BLOCK

(* This is a template for a factory with an heap based extendable memory pool {attribute 'hide_all_locals'} {attribute 'conditionalshow_all_locals' := 'SomeText'} {attribute 'conditionalshow_all_locals'} {attribute 'conditionalshow' := 'SomeText'} {attribute 'conditionalshow'} {attribute 'hide'} *)
{attribute 'enable_dynamic_creation'}
FUNCTION_BLOCK CustomFBFactory_heap EXTENDS FBF.FactoryBase

            SUPER^();

          

(* Please replace CustonFB with your specific function block type There is no need to change anything else !!! *)
METHOD Create : POINTER TO CustomFB
  VAR_INPUT
    itfData : FBF.IData;
  END_VAR
  VAR_OUTPUT
    eError : FBF.ERROR;
  END_VAR
  VAR
    hInst : CAA.HANDLE;
    itfInst : FBF.IInstance;
    xOk : BOOL;
  END_VAR
                  (* !!! This code must not be subject to change !!! *)
                      hInst := SUPER^.prvAllocInstMem(eError => eError);
                      Create := SUPER^.prvGetInstPointer(hInst);
                      IF Create <> 0 AND eError = FBF.ERROR.NO_ERROR THEN

                        {implicit on}
                        Create^.__vfInit();
                        Create^.FB_Init(TRUE, FALSE);
                        {implicit off}

                        xOk := __QUERYINTERFACE(Create^, itfInst);
                        IF xOk THEN
                          xOk := SUPER^.prvInstInit(itfInst, hInst, itfData, eError=>eError);
                        ELSE
                          eError := FBF.ERROR.WRONG_INTERFACE;
                        END_IF

                        IF NOT xOk THEN
                          SUPER^.prvFreeInstMem(hInst);
                          Create := CAA.gc_pNULL;
                        END_IF
                      END_IF
                    
                
END_METHOD
END_FUNCTION_BLOCK

(* This is a template for a factory with an static iec memory based memory pool which a fixed capacity {attribute 'hide_all_locals'} {attribute 'conditionalshow_all_locals' := 'SomeText'} {attribute 'conditionalshow_all_locals'} {attribute 'conditionalshow' := 'SomeText'} {attribute 'conditionalshow'} {attribute 'hide'} *)
{attribute 'enable_dynamic_creation'}
FUNCTION_BLOCK CustomFBFactory_static EXTENDS FBF.FactoryBase
  VAR
    abyPoolMemory : ARRAY[0..529] OF BYTE;  (* Please change the size of abyPoolMemory with your specific application need *)
  END_VAR

            SUPER^();

          

(* Please replace CustonFB with our specific function block type There is no need to change anything else !!! *)
METHOD Create : POINTER TO CustomFB
  VAR_INPUT
    itfData : FBF.IData;
  END_VAR
  VAR_OUTPUT
    eError : FBF.ERROR;
  END_VAR
  VAR
    hInst : CAA.HANDLE;
    itfInst : FBF.IInstance;
    xOk : BOOL;
  END_VAR
                  (* !!! This code must not be subject to change !!! *)
hInst := SUPER^.prvAllocInstMem(eError => eError);
Create := SUPER^.prvGetInstPointer(hInst);
IF Create <> 0 AND eError = FBF.ERROR.NO_ERROR THEN

	{implicit on}
	Create^.__vfInit();
	Create^.FB_Init(TRUE, FALSE);
	{implicit off}

	xOk := __QUERYINTERFACE(Create^, itfInst);
	IF xOk THEN
		xOk := SUPER^.prvInstInit(itfInst, hInst, itfData, eError=>eError);
	ELSE
		eError := FBF.ERROR.WRONG_INTERFACE;
	END_IF

	IF NOT xOk THEN
		SUPER^.prvFreeInstMem(hInst);
		Create := CAA.gc_pNULL;
	END_IF
END_IF
                
END_METHOD
END_FUNCTION_BLOCK
